{attribute addProperty BoxType "EL5101-0000-0001"}
{attribute addProperty Id "CtrlAT %Q*USINT811ValueAT %Q*UINT1622"}
{attribute addProperty CRC "1296992566"}
{attribute addProperty SizeInBites "24"}
{attribute addProperty SizeInBytes "3"}
TYPE Outputs_4D4E8936 :
STRUCT
	{attribute addProperty Name "Ctrl"}
	Ctrl AT %Q* : USINT;
	{attribute addProperty Name "Value"}
	Value AT %Q* : UINT;
END_STRUCT
END_TYPE

(* stored: Version 1.2.0.0, ProductVersion 3.1.4024.9
   DUT Outputs_4D4E8936: Id {dd3fae01-148a-42f0-a5b7-b9b419d8530b} *)
